// TwinCAT 3 PLC project UserMagExT_PLC
// ProgramVersion: 3.1.4023.0
// libraries:
//   Tc2_Standard, * (Beckhoff Automation GmbH)
//   Tc2_System, * (Beckhoff Automation GmbH)
//   Tc3_Module, * (Beckhoff Automation GmbH)
//   VisuDialogs, * (System)
//   VisuSymbols,3.5.10.0,System
// project tree:
//   DUTs/ ST_User.TcDUT
//   / GlobalTextList.TcGTLO, PlcTask.TcTTO, Visualization Manager.TcVMO (not stored), VISU_TASK.TcTTO
//   POUs/ MAIN.TcPOU, P_ListUsers.TcPOU, P_LoginFromPLC.TcPOU, P_TrackRemainingTime.TcPOU
//   VISUs/ CustomLoginDialog.TcVIS, Visualization.TcVIS
// real-time tasks:
//   TASK PlcTask: cycle T#10ms, priority 20, ADS port 350
//   TASK VISU_TASK: cycle T#200000us, priority 30, ADS port 351

CONFIGURATION UserMagExT_PLC
    RESOURCE PLC ON TwinCAT3
        TASK PlcTask(INTERVAL := T#10ms, PRIORITY := 20);
        TASK VISU_TASK(INTERVAL := T#200000us, PRIORITY := 30);
        PROGRAM MAIN WITH PlcTask : MAIN;
        PROGRAM VisuElems_Visu_Prg WITH VISU_TASK : VisuElems.Visu_Prg;
    END_RESOURCE
END_CONFIGURATION

// ---- DUTs/ST_User.TcDUT
TYPE ST_User :
STRUCT
	wsUserName		 	: WSTRING;
	wsUserFullName	 	: WSTRING;
	dwGroupID			: DWORD;
	bDeactivated		: BOOL;
END_STRUCT
END_TYPE

// ---- POUs/MAIN.TcPOU
PROGRAM MAIN
VAR
	bButton : BOOL;
END_VAR

P_TrackRemainingTime();
P_LoginFromPLC();
P_ListUsers();

END_PROGRAM

// ---- POUs/P_TrackRemainingTime.TcPOU
// przykladowy program sledzacy ile czasu zostalo do automatycznego wylogowwania danego uzytkownika
PROGRAM P_TrackRemainingTime
VAR
	aCurrentUser	:	ARRAY [0..2,0..10] OF WSTRING;	
	uiIndex			:	UINT;

	pClient			:	POINTER TO VisuElems.VisuElemBase.VisuStructClientData;
	sName			:	WSTRING;

// PWD for all users: "1"
	tHelp 			: TIME;
END_VAR

uiIndex := 0;

VisuElems.VisuElemBase.g_ClientManager.BeginIteration();

WHILE (pClient := VisuElems.VisuElemBase.g_ClientManager.GetNextClient()) <> 0 DO
	IF uiIndex < 10 THEN
		sName := pClient^.GlobalData.CurrentUserName;
		IF NOT (sName = "") THEN
			aCurrentUser[0,uiIndex] := sName;	

			IF pClient^.GlobalData.ClientType = VisuElems.VisuElemBase.Visu_ClientType.ProgrammingSystem THEN		
				aCurrentUser[1,uiIndex] := "ProgrammingSystem";
			ELSIF pClient^.GlobalData.ClientType = VisuElems.VisuElemBase.Visu_ClientType.WebVisualization THEN
				aCurrentUser[1,uiIndex] := "WebVisu";
			ELSE
				aCurrentUser[1,uiIndex] := "TargetVisu";
			END_IF	
			tHelp := pClient^.GlobalData.LastUsage - pClient^.GlobalData.AutoLogoutTimeStart;
			aCurrentUser[2,uiIndex] := TIME_TO_WSTRING(pClient^.GlobalData.AutoLogoutTime - tHelp);
		ELSE
			aCurrentUser[0,uiIndex] := "";
			aCurrentUser[1,uiIndex] := "";	
			aCurrentUser[2,uiIndex] := "";	
		END_IF
	END_IF
	uiIndex := uiIndex + 1;
END_WHILE

END_PROGRAM

// ---- POUs/P_LoginFromPLC.TcPOU
// przykalodwy program logujacy uzytkownika wizualizacji z poziomu kodu PLC
PROGRAM P_LoginFromPLC
VAR
	bLogIn 		: BOOL;
	pClient		: POINTER TO VisuElems.VisuStructClientData; 
END_VAR

IF bLogIn THEN
	VisuElems.g_ClientManager.BeginIteration(); 
	pClient := VisuElems.g_ClientManager.GetNextClient(); 
	
	WHILE pClient <> VisuElems.NULL DO 
		IF (pClient^.GlobalData.CurrentUserGroupId <> 1) THEN 
			VisuUserManagement.g_VisuUserMgmt2.LoginToUserGroup(pClient, 1, "Admin", "Administrator");
		END_IF 
		pClient := VisuElems.g_ClientManager.GetNextClient(); 
	END_WHILE
END_IF

END_PROGRAM

// ---- POUs/P_ListUsers.TcPOU
// program do odczytania danych o istniejacyhc uzytkownikach
PROGRAM P_ListUsers
VAR
	fbUserMng   			: VisuUserManagement.VisuUserMgmt;
   	stRet      				: VisuUserManagement.VUM_ReturnValues;
   	udiNumberOfUsers   		: UDINT;
   	dwUserDB         		: DWORD;
   	bUpdateUserList   		: BOOL;
   	aUserList         		: ARRAY[0..5] OF VisuUserManagement.VUM_User;
	aUsers					: ARRAY[0..2] OF ST_user; 
END_VAR

IF bUpdateUserList THEN
	bUpdateUserList:=FALSE;
   	dwUserDB := fbUserMng.GetUserDBAsCopy();
   	udiNumberOfUsers := fbUserMng.GetUserCount(dwUserDB);

 	stRet := fbUserMng.GetUsers(
                 dwUserDB:= dwUserDB, 
                 udiStartIndex:= 0, 
                 udiEndIndex:= udiNumberOfUsers-1, 
                 pArr:=  ADR(aUserList),
                 udiArrSize:= udiNumberOfUsers);
END_IF

A_Users();

ACTION A_Users:
//przepisanie pobranej listy uzytkownikow do tablicy ktora bedzie wuswietlana na wizualizacji

aUsers[0].wsUserName:=aUserList[0].wstUserName;
aUsers[0].wsUserFullName:=aUserList[0].wstFullName;
aUsers[0].dwGroupID:=aUserList[0].dwUserGroupID;
aUsers[0].bDeactivated:=aUserList[0].bDeactivated;

aUsers[1].wsUserName:=aUserList[1].wstUserName;
aUsers[1].wsUserFullName:=aUserList[1].wstFullName;
aUsers[1].dwGroupID:=aUserList[1].dwUserGroupID;
aUsers[1].bDeactivated:=aUserList[1].bDeactivated;

aUsers[2].wsUserName:=aUserList[2].wstUserName;
aUsers[2].wsUserFullName:=aUserList[2].wstFullName;
aUsers[2].dwGroupID:=aUserList[2].dwUserGroupID;
aUsers[2].bDeactivated:=aUserList[2].bDeactivated;
END_ACTION

END_PROGRAM

// ---- GlobalTextList.TcGTLO
TEXTLIST GlobalTextList
  880 = '%s'
  483 = '*'
  332 = '*****'
  973 = 'Access rights'
  107 = 'Admin'
  624 = 'Admin: operable'
  9 = 'Auto-fill username'
  744 = 'Be careful with this part, when adding users, adjust array size in program code'
  302 = 'Beckhoff Custom Login'
  334 = 'Cancel'
  66 = 'Change password (Admin)'
  300 = 'Current user group:'
  942 = 'Current user name:'
  742 = 'Deactiated'
  628 = 'Full Name'
  814 = 'Group ID'
  825 = 'Label'
  328 = 'LOGIN'
  214 = 'Login'
  355 = 'Login form PLC'
  169 = 'Login from PLC'
  200 = 'Logout'
  940 = 'LOGOUT'
  518 = 'Name'
  410 = 'None'
  333 = 'Ok'
  379 = 'Operator'
  344 = 'Operator: invisible'
  93 = 'Operator: visible'
  908 = 'Password for all users: 1'
  330 = 'Password:'
  520 = 'Remaining Logout Time'
  804 = 'Remaining time'
  661 = 'Service'
  544 = 'Service: visible'
  855 = 'Time'
  519 = 'Type'
  76 = 'Update'
  16 = 'User mngmt (Admin)'
  329 = 'User name:'
  438 = 'UserName'
  885 = 'Users list'
END_TEXTLIST

// ---- VISUs/CustomLoginDialog.TcVIS
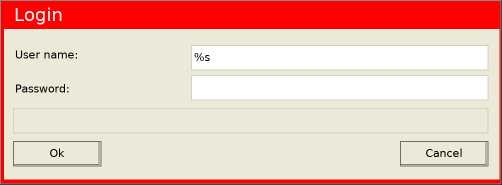
VISUALIZATION CustomLoginDialog  // 502x185
VAR
	iIndexLoginProvider : DWORD;
END_VAR
    Rectangle (0,0 502x185)
    Rectangle (4,29 495x150)
    Rectangle (11,0 476x30), "Login"
    Label (12,40 180x30), "User name:"
    Label (12,74 180x30), "Password:"
    Textfield (191,45 297x25), "%s", text variable: VisuUserManagement.g_VisuLoginProviderManager.m_arrLoginProvider[iIndexLoginProvider].stUserName
        OnMouseDown: write the text variable via Default
    Textfield (191,75 297x25), text variable: VisuUserManagement.g_VisuLoginProviderManager.m_arrLoginProvider[iIndexLoginProvider].stPassword
        OnMouseDown: write the text variable via Default, password
    Textfield (13,108 475x25), text list: '.VisuUserManagement.TL_VUM_Errors', text index: VisuUserManagement.g_VisuLoginProviderManager.m_arrLoginProvider[iIndexLoginProvider].udiLastError
    Button (13,141 88x25), "Ok"
        OnMouseDown: execute { VisuUserManagement.g_VisuLoginProviderManager.m_arrLoginProvider[iIndexLoginProvider].dwDialogResultOK := TRUE; }
    Button (400,141 88x25), "Cancel"
        OnMouseDown: execute { VisuUserManagement.g_VisuLoginProviderManager.m_arrLoginProvider[iIndexLoginProvider].dwDialogResultCancel := TRUE; }
END_VISUALIZATION

// ---- VISUs/Visualization.TcVIS
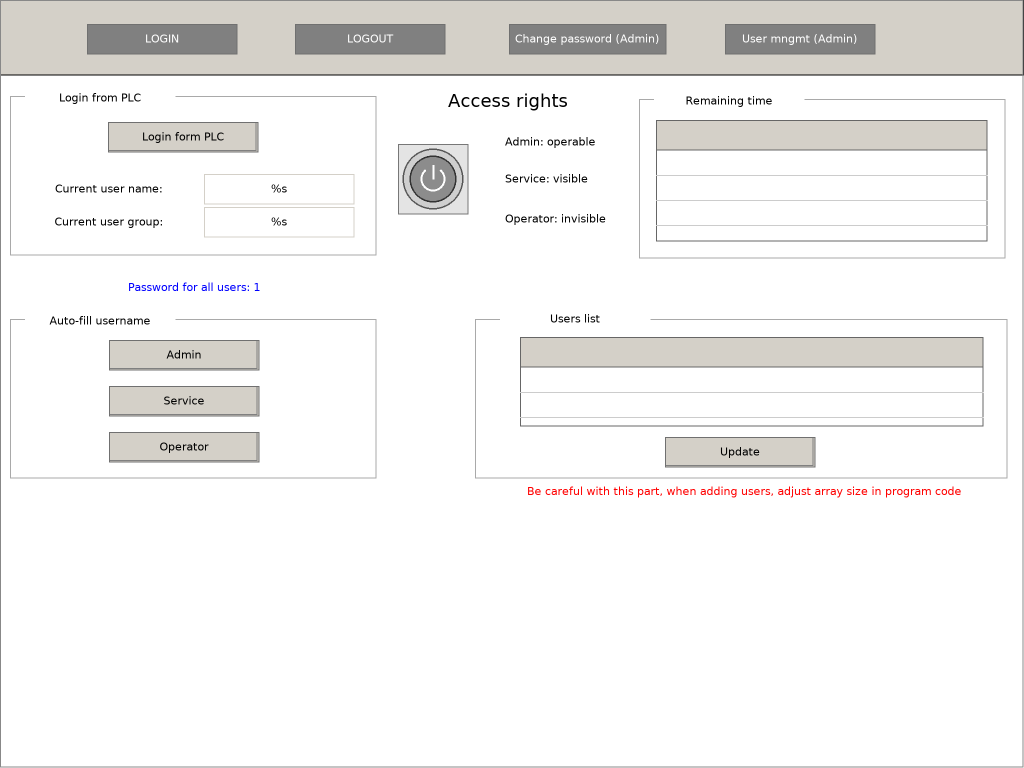
VISUALIZATION Visualization  // 1024x768
    Rectangle (10,319 366x159)
    Rectangle (639,99 366x159)
    Rectangle (0,0 1024x75)
    Button (87,24 150x30), "LOGIN"
        OnMouseDown: VisuUserMgmt Type=Login
    Button (295,24 150x30), "LOGOUT"
        OnMouseDown: VisuUserMgmt Type=Logout
    Button (509,24 157x30), "Change password (Admin)"
        OnMouseDown: VisuUserMgmt Type=ChangeUserPassword
    Button (725,24 150x30), "User mngmt (Admin)"
        OnMouseDown: VisuUserMgmt Type=OpenUserConfiguration
    Table (656,120 331x121), data array: P_TrackRemainingTime.aCurrentUser
        p3854506369: P_TrackRemainingTime.aCurrentUser[0,INDEX]
        p1892666644: P_TrackRemainingTime.aCurrentUser[1,INDEX]
        p338671338: P_TrackRemainingTime.aCurrentUser[2,INDEX]
        p2232123230: Name
        p511219082: Type
    Rectangle (654,86 150x30), "Remaining time"
    Rectangle (10,96 366x159)
    Rectangle (25,83 150x30), "Login from PLC"
    Button (108,122 150x30), "Login form PLC"
        tap P_LoginFromPLC.bLogIn
    Label (34,174 150x30), "Current user name:"
    Textfield (204,174 150x30), "%s", text variable: VisuElemsWinControls.CurrentUserName
    Rectangle (433,86 150x30), "Access rights"
    PowerSwitch (398,144 70x70), variable: MAIN.bButton, behaviour: TOGGLE, style: Switch-PowerSwitch-Gray
    Label (502,127 130x30), "Admin: operable"
    Label (502,164 130x30), "Service: visible"
    Label (502,204 130x30), "Operator: invisible"
    Rectangle (25,306 150x30), "Auto-fill username"
    Label (34,207 150x30), "Current user group:"
    Textfield (204,207 150x30), "%s", text variable: VisuElemsWinControls.CurrentUserGroupName
    Rectangle (475,319 532x159)
    Table (520,337 463x89), data array: P_ListUsers.aUsers
        p3854506369: P_ListUsers.aUsers[INDEX].wsUserName
        p1892666644: P_ListUsers.aUsers[INDEX].wsUserFullName
        p338671338: P_ListUsers.aUsers[INDEX].dwGroupID
        p2170511999: P_ListUsers.aUsers[INDEX].bDeactivated
        p511219082: Full Name
        p1755163831: Group ID
        p4092479075: Deactiated
    Rectangle (500,304 150x30), "Users list"
    Button (665,437 150x30), "Update"
        tap P_ListUsers.bUpdateUserList
    Label (483,463 523x57), "Be careful with this part, when adding users, adjust array size in program code"
    Label (13,259 363x57), "Password for all users: 1"
    Button (109,340 150x30), "Admin", colour toggle: VisuElemsWinControls.CurrentUserName="Admin"
        OnMouseDown: VisuUserMgmt Type=Login
        OnMouseDown: execute { VisuUserManagement.g_VisuLoginProviderManager.m_arrLoginProvider[0].stUserName := "Admin"; }
    Button (109,386 150x30), "Service", colour toggle: VisuElemsWinControls.CurrentUserName="Service"
        OnMouseDown: VisuUserMgmt Type=Login
        OnMouseDown: execute { VisuUserManagement.g_VisuLoginProviderManager.m_arrLoginProvider[0].stUserName := "Service"; }
    Button (109,432 150x30), "Operator", colour toggle: VisuElemsWinControls.CurrentUserName="Operator"
        OnMouseDown: VisuUserMgmt Type=Login
        OnMouseDown: execute { VisuUserManagement.g_VisuLoginProviderManager.m_arrLoginProvider[0].stUserName := "Operator"; }
END_VISUALIZATION
